Staubli VAL3: GetArrayIndex.pgx

public program GetArrayIndex(string& x_In[], string x_sFindStr, num x_nSelect, num& x_nIndex)
  local num l_i
begin
  //查找x_sFindStr在x_In中细分类别的索引值
  //x_nSelect:x_In中的第x_nSelect+1个元素
  //找到返回x_Index,否则返回-1
  //例如：x_In=[0，a],[1，a],[3,b],[4,a],[5,b],[6,b];x_nSelect=3
  //因为x_In由[0,a],[1,a],[4,a]和[3,b],[5,b],[6,b]
  //当x_nSelect=3时，对x_In为[3,b]，而该值在[b]值为第一个，故 x_nIndex=0；
  x_nIndex=-1
  if x_nSelect>size(x_In)
    x_nSelect=size(x_In)-1
  endIf
  for l_i=0 to x_nSelect
    if find(x_In[l_i],x_sFindStr)!=-1
      x_nIndex=x_nIndex+1
    endIf
  endFor
end
